// TwinCAT 3 PLC project Untitled1
// ProgramVersion: 3.1.4024.0
// libraries:
//   CmpBitmapPool, * (System)
//   Tc2_Standard, * (Beckhoff Automation GmbH)
//   Tc2_System, * (Beckhoff Automation GmbH)
//   Tc3_Module, * (Beckhoff Automation GmbH)
//   TwinCAT_LIB, * (Farnwood Engineering)
// project tree:
//   / PlcTask.TcTTO
//   POUs/2. Equipment Modules/1. EM_Can_Supply/ FB_Can_Supply.TcPOU, E_State_Can_Supply.TcDUT, ITF_Can_Supply.TcIO, Str_fb_mem.TcDUT
//   POUs/2. Equipment Modules/2. EM_OutfeedA/ EM_OutfeedA.TcPOU
//   POUs/2. Equipment Modules/3. EM_OutfeedA2/ EM_OutfeedA2.TcPOU
//   POUs/3. Units/Unit_Blikkenvullijn/ ITF_Blikkenvullijn.TcIO, UNIT_Blikkenvullijn.TcPOU
//   POUs/ FB_DevicesV2.TcPOU, MAIN.TcPOU
// real-time tasks:
//   TASK PlcTask: cycle T#10ms, priority 20, ADS port 350

CONFIGURATION Untitled1
    RESOURCE PLC ON TwinCAT3
        TASK PlcTask(INTERVAL := T#10ms, PRIORITY := 20);
        PROGRAM MAIN WITH PlcTask : MAIN;
    END_RESOURCE
END_CONFIGURATION

// ---- POUs/2. Equipment Modules/1. EM_Can_Supply/E_State_Can_Supply.TcDUT
{attribute 'qualified_only'}
{attribute 'strict'}
TYPE E_State_Can_Supply :
(
	State := 0
);
END_TYPE

// ---- POUs/2. Equipment Modules/1. EM_Can_Supply/Str_fb_mem.TcDUT
TYPE Str_fb_mem :
STRUCT
	State : E_State_PackML;
END_STRUCT
END_TYPE

// ---- POUs/2. Equipment Modules/1. EM_Can_Supply/ITF_Can_Supply.TcIO
INTERFACE ITF_Can_Supply EXTENDS ITF_PackML

END_INTERFACE

// ---- POUs/3. Units/Unit_Blikkenvullijn/ITF_Blikkenvullijn.TcIO
INTERFACE ITF_Blikkenvullijn

END_INTERFACE

// ---- POUs/MAIN.TcPOU
PROGRAM MAIN
VAR
	Unit : UNIT_Blikkenvullijn;
	Devices : FB_DevicesV2;
END_VAR

(*
$$$$$$$$\                                                                   $$\       $$$$$$$$\                     $$\                                         $$\                     
$$  _____|                                                                  $$ |      $$  _____|                    \__|                                        \__|                    
$$ |   $$$$$$\   $$$$$$\  $$$$$$$\  $$\  $$\  $$\  $$$$$$\   $$$$$$\   $$$$$$$ |      $$ |      $$$$$$$\   $$$$$$\  $$\ $$$$$$$\   $$$$$$\   $$$$$$\   $$$$$$\  $$\ $$$$$$$\   $$$$$$\  
$$$$$\ \____$$\ $$  __$$\ $$  __$$\ $$ | $$ | $$ |$$  __$$\ $$  __$$\ $$  __$$ |      $$$$$\    $$  __$$\ $$  __$$\ $$ |$$  __$$\ $$  __$$\ $$  __$$\ $$  __$$\ $$ |$$  __$$\ $$  __$$\ 
$$  __|$$$$$$$ |$$ |  \__|$$ |  $$ |$$ | $$ | $$ |$$ /  $$ |$$ /  $$ |$$ /  $$ |      $$  __|   $$ |  $$ |$$ /  $$ |$$ |$$ |  $$ |$$$$$$$$ |$$$$$$$$ |$$ |  \__|$$ |$$ |  $$ |$$ /  $$ |
$$ |  $$  __$$ |$$ |      $$ |  $$ |$$ | $$ | $$ |$$ |  $$ |$$ |  $$ |$$ |  $$ |      $$ |      $$ |  $$ |$$ |  $$ |$$ |$$ |  $$ |$$   ____|$$   ____|$$ |      $$ |$$ |  $$ |$$ |  $$ |
$$ |  \$$$$$$$ |$$ |      $$ |  $$ |\$$$$$\$$$$  |\$$$$$$  |\$$$$$$  |\$$$$$$$ |      $$$$$$$$\ $$ |  $$ |\$$$$$$$ |$$ |$$ |  $$ |\$$$$$$$\ \$$$$$$$\ $$ |      $$ |$$ |  $$ |\$$$$$$$ |
\__|   \_______|\__|      \__|  \__| \_____\____/  \______/  \______/  \_______|      \________|\__|  \__| \____$$ |\__|\__|  \__| \_______| \_______|\__|      \__|\__|  \__| \____$$ |
                                                                                                          $$\   $$ |                                                          $$\   $$ |
                                                                                                          \$$$$$$  |                                                          \$$$$$$  |
                                                                                                           \______/                                                            \______/ 
*)

//*****************************UNIT*****************************//
Unit();

//******************************CM******************************//
Devices();

END_PROGRAM

// ---- POUs/3. Units/Unit_Blikkenvullijn/UNIT_Blikkenvullijn.TcPOU
FUNCTION_BLOCK UNIT_Blikkenvullijn IMPLEMENTS  ITF_Blikkenvullijn
VAR
	EM_Can_Supply 		: FB_Can_Supply;
	EM_Filling			: FB_Machine_PackML;
	EM_Check_Weigher	: FB_Machine_PackML;
	EM_Labeller			: FB_Machine_PackML;
	EM_Turning			: FB_Machine_PackML;
	EM_Stamp			: FB_Machine_PackML;
	EM_Seal_Shrink		: FB_Machine_PackML;
END_VAR

(*
$$$$$$$$\                                                                   $$\       $$$$$$$$\                     $$\                                         $$\                     
$$  _____|                                                                  $$ |      $$  _____|                    \__|                                        \__|                    
$$ |   $$$$$$\   $$$$$$\  $$$$$$$\  $$\  $$\  $$\  $$$$$$\   $$$$$$\   $$$$$$$ |      $$ |      $$$$$$$\   $$$$$$\  $$\ $$$$$$$\   $$$$$$\   $$$$$$\   $$$$$$\  $$\ $$$$$$$\   $$$$$$\  
$$$$$\ \____$$\ $$  __$$\ $$  __$$\ $$ | $$ | $$ |$$  __$$\ $$  __$$\ $$  __$$ |      $$$$$\    $$  __$$\ $$  __$$\ $$ |$$  __$$\ $$  __$$\ $$  __$$\ $$  __$$\ $$ |$$  __$$\ $$  __$$\ 
$$  __|$$$$$$$ |$$ |  \__|$$ |  $$ |$$ | $$ | $$ |$$ /  $$ |$$ /  $$ |$$ /  $$ |      $$  __|   $$ |  $$ |$$ /  $$ |$$ |$$ |  $$ |$$$$$$$$ |$$$$$$$$ |$$ |  \__|$$ |$$ |  $$ |$$ /  $$ |
$$ |  $$  __$$ |$$ |      $$ |  $$ |$$ | $$ | $$ |$$ |  $$ |$$ |  $$ |$$ |  $$ |      $$ |      $$ |  $$ |$$ |  $$ |$$ |$$ |  $$ |$$   ____|$$   ____|$$ |      $$ |$$ |  $$ |$$ |  $$ |
$$ |  \$$$$$$$ |$$ |      $$ |  $$ |\$$$$$\$$$$  |\$$$$$$  |\$$$$$$  |\$$$$$$$ |      $$$$$$$$\ $$ |  $$ |\$$$$$$$ |$$ |$$ |  $$ |\$$$$$$$\ \$$$$$$$\ $$ |      $$ |$$ |  $$ |\$$$$$$$ |
\__|   \_______|\__|      \__|  \__| \_____\____/  \______/  \______/  \_______|      \________|\__|  \__| \____$$ |\__|\__|  \__| \_______| \_______|\__|      \__|\__|  \__| \____$$ |
                                                                                                          $$\   $$ |                                                          $$\   $$ |
                                                                                                          \$$$$$$  |                                                          \$$$$$$  |
                                                                                                           \______/                                                            \______/ 
*)

//**************************INITIATE**************************//
//*****************************EM*****************************//
//*************************BlackBoxes*************************//
EM_Filling();
EM_Check_Weigher();
EM_Labeller();
EM_Turning();
EM_Stamp();
EM_Seal_Shrink();
//*************************Custommade*************************//
EM_Can_Supply();

METHOD FB_init : BOOL
VAR_INPUT
	bInitRetains : BOOL; // if TRUE, the retain variables are initialized (warm start / cold start)
	bInCopyCode : BOOL;  // if TRUE, the instance afterwards gets moved into the copy code (online change)
END_VAR
//*****************************INITIATE*****************************//
EM_Can_Supply.FB_init(0,0);
EM_Filling.FB_init(0,0);
EM_Check_Weigher.FB_init(0,0);
EM_Labeller.FB_init(0,0);
EM_Turning.FB_init(0,0);
EM_Stamp.FB_init(0,0);
EM_Seal_Shrink.FB_init(0,0);
END_METHOD

END_FUNCTION_BLOCK

// ---- POUs/2. Equipment Modules/1. EM_Can_Supply/FB_Can_Supply.TcPOU
FUNCTION_BLOCK FB_Can_Supply IMPLEMENTS  ITF_Can_Supply
VAR
	fb_mem : Str_fb_mem;
	PackML : FB_PackML;
END_VAR

(*
$$$$$$$$\                                                                   $$\       $$$$$$$$\                     $$\                                         $$\                     
$$  _____|                                                                  $$ |      $$  _____|                    \__|                                        \__|                    
$$ |   $$$$$$\   $$$$$$\  $$$$$$$\  $$\  $$\  $$\  $$$$$$\   $$$$$$\   $$$$$$$ |      $$ |      $$$$$$$\   $$$$$$\  $$\ $$$$$$$\   $$$$$$\   $$$$$$\   $$$$$$\  $$\ $$$$$$$\   $$$$$$\  
$$$$$\ \____$$\ $$  __$$\ $$  __$$\ $$ | $$ | $$ |$$  __$$\ $$  __$$\ $$  __$$ |      $$$$$\    $$  __$$\ $$  __$$\ $$ |$$  __$$\ $$  __$$\ $$  __$$\ $$  __$$\ $$ |$$  __$$\ $$  __$$\ 
$$  __|$$$$$$$ |$$ |  \__|$$ |  $$ |$$ | $$ | $$ |$$ /  $$ |$$ /  $$ |$$ /  $$ |      $$  __|   $$ |  $$ |$$ /  $$ |$$ |$$ |  $$ |$$$$$$$$ |$$$$$$$$ |$$ |  \__|$$ |$$ |  $$ |$$ /  $$ |
$$ |  $$  __$$ |$$ |      $$ |  $$ |$$ | $$ | $$ |$$ |  $$ |$$ |  $$ |$$ |  $$ |      $$ |      $$ |  $$ |$$ |  $$ |$$ |$$ |  $$ |$$   ____|$$   ____|$$ |      $$ |$$ |  $$ |$$ |  $$ |
$$ |  \$$$$$$$ |$$ |      $$ |  $$ |\$$$$$\$$$$  |\$$$$$$  |\$$$$$$  |\$$$$$$$ |      $$$$$$$$\ $$ |  $$ |\$$$$$$$ |$$ |$$ |  $$ |\$$$$$$$\ \$$$$$$$\ $$ |      $$ |$$ |  $$ |\$$$$$$$ |
\__|   \_______|\__|      \__|  \__| \_____\____/  \______/  \______/  \_______|      \________|\__|  \__| \____$$ |\__|\__|  \__| \_______| \_______|\__|      \__|\__|  \__| \____$$ |
                                                                                                          $$\   $$ |                                                          $$\   $$ |
                                                                                                          \$$$$$$  |                                                          \$$$$$$  |
                                                                                                           \______/                                                            \______/ 
*)

//EXTERNE STATE CHANGES
IF 



// INTERNAL STATE CHANGES
IF PackML.State.get() = E_State_PackML.IDLE THEN
	// Do nothing
END_IF

IF fb_mem.State = E_State_PackML.STARTING THEN
	Starting_SC := TRUE;
END_IF

IF fb_mem.State = E_State_PackML.EXECUTE THEN
	
	Execute_SC := TRUE;
END_IF

IF fb_mem.State = E_State_PackML.Completing THEN
	Completing_SC := TRUE;
END_IF

IF fb_mem.State = E_State_PackML.Complete THEN
	//Do nothing
END_IF

IF fb_mem.State = E_State_PackML.Resetting THEN
	Resetting_SC := TRUE;
END_IF

IF fb_mem.State = E_State_PackML.Holding THEN
	Holding_SC := TRUE;
END_IF

IF fb_mem.State = E_State_PackML.Held THEN
	Unholding_SC := TRUE;
END_IF

IF fb_mem.State = E_State_PackML.Unholding THEN
	Unholding_SC := TRUE;
END_IF

IF fb_mem.State = E_State_PackML.Suspending THEN
	Suspending_SC := TRUE;
END_IF

IF fb_mem.State = E_State_PackML.Suspended THEN
	//Do nothing
END_IF

IF fb_mem.State = E_State_PackML.Unsuspending THEN
	Unsuspending_SC := TRUE;
END_IF

IF fb_mem.State = E_State_PackML.Aborting THEN
	Aborting_SC := TRUE;
END_IF

IF fb_mem.State = E_State_PackML.Aborted THEN
	Clearing_SC := TRUE;
END_IF

IF fb_mem.State = E_State_PackML.Clearing THEN
	Clearing_SC := TRUE;
END_IF

IF fb_mem.State = E_State_PackML.Stopping THEN
	Stopping_SC := TRUE;
END_IF

IF fb_mem.State = E_State_PackML.Stopped THEN
	//Do nothing
END_IF

{error 'add property implementation or delete property to use base implementation'}
PROPERTY State : E_State_Can_Supply
GET
END_GET
END_PROPERTY

END_FUNCTION_BLOCK

// ---- POUs/FB_DevicesV2.TcPOU
FUNCTION_BLOCK FB_DevicesV2 

VAR

END_VAR

//INITIEREN

//Kleppen

//Object dat het waterpeil berekend


//Object wat een gewenst debiet kan simuleren


//Object dat de kleppen regelt

END_FUNCTION_BLOCK

// ---- POUs/2. Equipment Modules/2. EM_OutfeedA/EM_OutfeedA.TcPOU
FUNCTION_BLOCK EM_OutfeedA EXTENDS FB_Transport
VAR_INPUT
END_VAR
VAR_OUTPUT
END_VAR
VAR
END_VAR

//Thijs is gejoined
//Thijs is opnieuw gejoined

END_FUNCTION_BLOCK

// ---- POUs/2. Equipment Modules/3. EM_OutfeedA2/EM_OutfeedA2.TcPOU
FUNCTION_BLOCK EM_OutfeedA2 EXTENDS FB_Transport
FUNCTION_BLOCK EM_OutfeedA2 EXTENDS FB_Mechanische_Stop

VAR
	fb_mem : Str_FB_Transport;
END_VAR

END_FUNCTION_BLOCK
